// TIA Portal V20 export
// export: Created 2025-12-01T14:57:27.4021736Z, ExportSetting None, DisplayName Totally Integrated Automation Portal, DisplayVersion V20 Update 3, DisplayName TIA Portal Openness, DisplayVersion V20 Update 3, DisplayName TIA Portal Version Control Interface, DisplayVersion V20 Update 3, DisplayName STEP 7 Professional, DisplayVersion V20 Update 3, DisplayName STEP 7 Safety, DisplayVersion V20 Update 2, DisplayName WinCC Basic/Comfort/Advanced, DisplayVersion V20 Update 3, DisplayName WinCC Professional, DisplayVersion V20 Update 3, DisplayName WinCC Unified, DisplayVersion V20 Update 3
FUNCTION_BLOCK "FB607_SalidaMovil_Frontal_Quimarox"   // FB607, LAD
{ S7_Optimized_Access := 'FALSE' }
// stored: AutoNumber false, SetENOAutomatically false
   VAR_INPUT
      MesaDeDescarga : UInt;
      ID_Quimarox : UInt;
      ID_Elemento : UInt;
      DestinoAsociado : UInt;
      pHs_PosicionDescarga : Bool;
      pHs_Protrusion : Bool;
      En_PosicionReposo : Bool;
      Corte_PosicionReposo : Bool;
      Corte_PosicionDesCarga : Bool;
      En_PosicionDescarga : Bool;
      Permiso_DeDesCarga : Bool;
      V_Filtro_pHsPresencia : Int;
      Pto_Ajuste_1 : Int;   // en mm (paso a lenta en posicionamiento a descarga de transportador)
      Pto_Ajuste_2 : Int;   // en mm (timeout movimiento posicion descarga del transportador)
      Pto_Ajuste_3 : Int;   // en mm (paso a lenta en posicionamiento reposo del transportador)
      Pto_Ajuste_4 : Int;   // en mm (timeout movimiento posicion reposo del transportador)
   END_VAR
   VAR_OUTPUT
      NXT_DescargaActiva : Bool;
      ElevadorEnLenta : Bool;
      PararElevador : Bool;
      Ir_PosicionReposo : Bool;
      Ir_PosicionDescarga : Bool;
   END_VAR
   VAR
      FILTRO_pHsPresencia : "FB910_CNT_UHS";
      EstadoAsociadoEnMesa : UInt;
      Ultimo_PeineTratado : UInt;
      Aux_PeineEnDesCarga { ExternalAccessible := 'False'; ExternalVisible := 'False'; ExternalWritable := 'False'} : UInt;
   END_VAR
   VAR_TEMP
      MesaQuimarox : UInt;
      NumeroUT : UInt;
      Vagon_Siguiente : Int;
      EsMesaTL : Bool;
      FILTRO_PosicionDesCarga : Bool;
   END_VAR
BEGIN

NETWORK
TITLE = ERROR - Rearme
/////////////////////////////////////////////////////////////
/////////////////////////////////////////////////////////////
/////////////////////////////////////////////////////////////
// Rearne de Errores
      SET;
      A     "DB902_Estado_ZonaMesa".EstadoMesas[#MesaDeDescarga].Rearme_CBx;
      O     "DB902_Estado_ZonaMesa".EstadoMesas[#MesaDeDescarga].PerReset_CBx;
      R     "DB900_Estado_Mesas".EstadoVI[#MesaDeDescarga].Error_Mx;
      R     "DB900_Estado_Mesas".EstadoVI[#MesaDeDescarga].Err_Protusion;
      R     "DB900_Estado_Mesas".EstadoVI[#MesaDeDescarga].Err_TOut_Avance_E1_E3;
      R     "DB900_Estado_Mesas".EstadoVI[#MesaDeDescarga].Err_Tout_Sacar;
      R     "DB900_Estado_Mesas".EstadoVI[#MesaDeDescarga].Err_Tout_Recoger;

      R     "DB900_Estado_Mesas".EstadoVI[#MesaDeDescarga].Err_DatosPLC;



NETWORK
TITLE = HMI - Entradas y Salidas de la Mesa
/////////////////////////////////////////////////////////////
/////////////////////////////////////////////////////////////
/////////////////////////////////////////////////////////////
// Entradas
      SET;
      A     #pHs_PosicionDescarga;
      =     "DB904_Estado_Maquinas".EstadoVI[#MesaDeDescarga].Byte7_bit4;
      SET;
      A     #pHs_Protrusion;
      =     "DB904_Estado_Maquinas".EstadoVI[#MesaDeDescarga].Byte9_bit0;

      SET;
      A     #En_PosicionReposo;
      =     "DB904_Estado_Maquinas".EstadoVI[#MesaDeDescarga].Byte8_bit4;
      SET;
      A     #Corte_PosicionReposo;
      =     "DB904_Estado_Maquinas".EstadoVI[#MesaDeDescarga].Byte7_bit6;
      SET;
      A     #Corte_PosicionDesCarga;
      =     "DB904_Estado_Maquinas".EstadoVI[#MesaDeDescarga].Byte7_bit7;
      SET;
      A     #En_PosicionDescarga;
      =     "DB904_Estado_Maquinas".EstadoVI[#MesaDeDescarga].Byte8_bit5;


// Salidas
      SET;
      A     #NXT_DescargaActiva;
      =     "DB900_Estado_Mesas".EstadoVI[#MesaDeDescarga].Sa_Giro_180;
      SET;
      A     #Ir_PosicionReposo;
      =     "DB900_Estado_Mesas".EstadoVI[#MesaDeDescarga].Sa_Trans_Baj;
      SET;
      A     #Ir_PosicionDescarga;
      =     "DB900_Estado_Mesas".EstadoVI[#MesaDeDescarga].Sa_Trans_Sub;



NETWORK
TITLE = Comprobacion de que la MESA es de TRACKING
/////////////////////////////////////////////////////////////////////////////////////
/////////////////////////////////////////////////////////////////////////////////////
/////////////////////////////////////////////////////////////////////////////////////
// Comprobar si es una Mesa de Tracking o Routing
      SET;
      A     "DB850_DefinicionMesas".Mesa[#MesaDeDescarga].ConfigMesa.MesaTL;
      =     #EsMesaTL;



NETWORK
TITLE = Inicializacio PREVIA
/////////////////////////////////////////////////////////////////////////////////////
/////////////////////////////////////////////////////////////////////////////////////
/////////////////////////////////////////////////////////////////////////////////////
      CLR;
      =     #ElevadorEnLenta;
      =     #PararElevador;

      CLR;
      =     #NXT_DescargaActiva;

      CLR;
      =     #Ir_PosicionReposo;
      =     #Ir_PosicionDescarga;



NETWORK
TITLE = SISTEMA - Reset
/////////////////////////////////////////////////////////////
/////////////////////////////////////////////////////////////
/////////////////////////////////////////////////////////////
// - Existe RESET ??
      SET;
      AN    "DB902_Estado_ZonaMesa".EstadoMesas[#MesaDeDescarga].PerReset_CBx;  //#Estado_CBx.PerReset_CBx
      JC    NoRealizandose_Reset;

      L     0;
      T     #EstadoAsociadoEnMesa;
      T     #Ultimo_PeineTratado;


/////////////////////////////////////////////////////////////
/////////////////////////////////////////////////////////////
/////////////////////////////////////////////////////////////
// - Final Tratamiento del RESET
NoRealizandose_Reset:NOP   0;



NETWORK
TITLE = >>>>>>>>>>>>>>>>>>>>>>>>>>>>>>>>>>>>>>>>>>>>>>>>>>>>>>>>>>>>>>>>>>>

REGION Network 7: FILTRO - pHs de Presencia
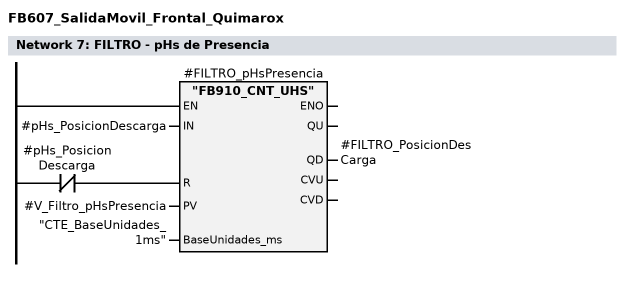
   RUNG wire#powerrail
      #FILTRO_pHsPresencia(R := wire#w1, IN := #pHs_PosicionDescarga, PV := #V_Filtro_pHsPresencia, BaseUnidades_ms := "CTE_BaseUnidades_1ms", QU =>, QD => #FILTRO_PosicionDesCarga, CVU =>, CVD =>)
   END_RUNG
   RUNG wire#powerrail
      I_Contact( #pHs_PosicionDescarga )
   END_RUNG wire#w1
   // the same network as SCL:
   #FILTRO_pHsPresencia(IN := #pHs_PosicionDescarga,   // "FB910_CNT_UHS"
                        R := NOT #pHs_PosicionDescarga,
                        PV := #V_Filtro_pHsPresencia,
                        BaseUnidades_ms := "CTE_BaseUnidades_1ms",
                        QD => #FILTRO_PosicionDesCarga);
END_REGION

NETWORK
TITLE = >>>>>>>>>>>>>>>>>>>>>>>>>>>>>>>>>>>>>>>>>>>>>>>>>>>>>>>>>>>>>>>>>>>

NETWORK
TITLE = Control Etapa activa >>> DISTRIBUCION
/////////////////////////////////////////////////////////////////////////////////////
/////////////////////////////////////////////////////////////////////////////////////
/////////////////////////////////////////////////////////////////////////////////////
// listado de saltos de programa
      L     #EstadoAsociadoEnMesa;

      JL    ETAPA_PorDefecto;
      JU    ETAPA_00_EnReset;
      JU    ETAPA_01_EnReposo;

      JU    ETAPA_02_EsperaPermisoDeDescarga;
      JU    ETAPA_03_MoverPosicionDescarga;
      JU    ETAPA_04_PreparadoParaDescarga;
      JU    ETAPA_05_FinDescarga;
      JU    ETAPA_06_MoverPosicionReposo;

      JU    ETAPA_PorDefecto;
      JU    ETAPA_PorDefecto;
      JU    ETAPA_PorDefecto;

      JU    ETAPA_10_ResetVacio_EsperaDesCargaDePeine;
      JU    ETAPA_11_ResetVacio_RecogerCargaDePeine;
      JU    ETAPA_12_ResetVacio_MoverPosicionReposo;
      JU    ETAPA_13_ResetCargado_EsperaPermisoDeDesCarga;
      JU    ETAPA_14_ResetCargado_MoverPosicionReposo;

ETAPA_PorDefecto:JU    FinFuncion;




NETWORK
TITLE = ETAPA 00 >>> En Reset
/////////////////////////////////////////////////////////////////////////////////////
/////////////////////////////////////////////////////////////////////////////////////
/////////////////////////////////////////////////////////////////////////////////////
ETAPA_00_EnReset:NOP   0;
      CLR;
      =     #Ir_PosicionReposo;
      =     #Ir_PosicionDescarga;

/////////////////////////////////////////////////////////////////////////////////////
// error de protusion
      SET;
      AN    #pHs_Protrusion;
      JC    ErrorProtrusion;

/////////////////////////////////////////////////////////////////////////////////////
// Tiene que estar en Marcha y Sin Error para continuar
      SET;
      AN    "DB902_Estado_ZonaMesa".EstadoMesas[#MesaDeDescarga].Marcha_CBx;
      O     "DB902_Estado_ZonaMesa".EstadoMesas[#MesaDeDescarga].Error_CBx;
      JC    ET00_PararElevador;


/////////////////////////////////////////////////////////////////////////////////////
// En Resposo
      SET;
      A     #En_PosicionReposo;
      JC    ET00_IrEtapa_01_EnReposo;


/////////////////////////////////////////////////////////////////////////////////////
// NO Reposo - Vacio
      SET;
      AN    #FILTRO_PosicionDesCarga;
      JC    ET00_Reset_10_ResetVacio_EsperaDesCargaDePeine;

/////////////////////////////////////////////////////////////////////////////////////
// NO Reposo - Con Carga
      SET;
      A     #FILTRO_PosicionDesCarga;
      JC    ET00_Reset_13_ResetCargado_EsperaPermisoDeDesCarga;


/////////////////////////////////////////////////////////////////////////////////////
// Final del Reparto  ?????? No DEBE LLEGAR AQUI
      BE;




/////////////////////////////////////////////////////////////////////////////////////
/////////////////////////////////////////////////////////////////////////////////////
/////////////////////////////////////////////////////////////////////////////////////
ET00_PararElevador:NOP   0;
      SET;
      =     #PararElevador;
      BE;


/////////////////////////////////////////////////////////////////////////////////////
/////////////////////////////////////////////////////////////////////////////////////
/////////////////////////////////////////////////////////////////////////////////////
ET00_IrEtapa_01_EnReposo:NOP   0;
      L     1;
      T     #EstadoAsociadoEnMesa;
      JU    ETAPA_01_EnReposo;


/////////////////////////////////////////////////////////////////////////////////////
/////////////////////////////////////////////////////////////////////////////////////
/////////////////////////////////////////////////////////////////////////////////////
ET00_Reset_10_ResetVacio_EsperaDesCargaDePeine:NOP   0;
      L     10;
      T     #EstadoAsociadoEnMesa;
      JU    ETAPA_10_ResetVacio_EsperaDesCargaDePeine;


/////////////////////////////////////////////////////////////////////////////////////
/////////////////////////////////////////////////////////////////////////////////////
/////////////////////////////////////////////////////////////////////////////////////
ET00_Reset_13_ResetCargado_EsperaPermisoDeDesCarga:NOP   0;
      L     13;
      T     #EstadoAsociadoEnMesa;
      JU    ETAPA_13_ResetCargado_EsperaPermisoDeDesCarga;



NETWORK
TITLE = ETAPA 01 >>> En Reposo
/////////////////////////////////////////////////////////////////////////////////////
/////////////////////////////////////////////////////////////////////////////////////
/////////////////////////////////////////////////////////////////////////////////////
// Estado de reposo esperando a que llegue una carga para este destino
ETAPA_01_EnReposo:NOP   0;
      SET;
      AN    #En_PosicionReposo;
      JC    ET01_IrEtapa_14_MoverPosicionReposo;

/////////////////////////////////////////////////////////////////////////////////////
// miramos si ya hemos comprobado el peine que está delante nuestro
      SET;
      L     "DB602_ElementosQuimarox".Quimarox[#ID_Quimarox].Elementos[#ID_Elemento].Numero_carrier;
      L     #Ultimo_PeineTratado;
      ==I;
      JC    ET01_SinPeineEnVentana;

/////////////////////////////////////////////////////////////////////////////////////
// si no hemos comprobado el peine, comprobamos si tenemos un peine en ventana
      SET;
      AN    "DB602_ElementosQuimarox".Quimarox[#ID_Quimarox].Elementos[#ID_Elemento].Hay_Carrier_en_ventana;
      JC    ET01_SinPeineEnVentana;

/////////////////////////////////////////////////////////////////////////////////////
// si no ha saltado es porque el carrier está en ventana. Comprobamos si es para nosotros
      L     "DB602_ElementosQuimarox".Quimarox[#ID_Quimarox].Elementos[#ID_Elemento].Numero_carrier;
      T     #Aux_PeineEnDesCarga;

      SET;
      L     "DB601_PeinesQuimarox".Quimarox[#ID_Quimarox].vagon[#Aux_PeineEnDesCarga].Destino_principal;
      L     #DestinoAsociado;
      ==I;
      JC    ET01_PeineParaLaMesa;

/////////////////////////////////////////////////////////////////////////////////////
// si no es para mi, me guardo que he chequeado el peine para no volver a comprobarlo
      L     "DB602_ElementosQuimarox".Quimarox[#ID_Quimarox].Elementos[#ID_Elemento].Numero_carrier;
      T     #Ultimo_PeineTratado;
      BE;


/////////////////////////////////////////////////////////////////////////////////////
/////////////////////////////////////////////////////////////////////////////////////
/////////////////////////////////////////////////////////////////////////////////////
ET01_SinPeineEnVentana:NOP   0;
      SET;  // Esta TOTALMENTE libre ?
      A(;
      O     #FILTRO_PosicionDesCarga;
      ON    #pHs_Protrusion;
      );
      JCN   FinFuncion;
      JU    ErrorProtrusion;


/////////////////////////////////////////////////////////////////////////////////////
/////////////////////////////////////////////////////////////////////////////////////
/////////////////////////////////////////////////////////////////////////////////////
ET01_PeineParaLaMesa:NOP   0;
      L     2;
      T     #EstadoAsociadoEnMesa;
      L     "DB602_ElementosQuimarox".Quimarox[#ID_Quimarox].Elementos[#ID_Elemento].Numero_carrier;
      T     #Ultimo_PeineTratado;

      JU    ETAPA_02_EsperaPermisoDeDescarga;


/////////////////////////////////////////////////////////////////////////////////////
/////////////////////////////////////////////////////////////////////////////////////
/////////////////////////////////////////////////////////////////////////////////////
ET01_IrEtapa_14_MoverPosicionReposo:NOP   0;
      L     14;
      T     #EstadoAsociadoEnMesa;
      JU    ETAPA_14_ResetCargado_MoverPosicionReposo;


NETWORK
TITLE = ETAPA 02 >>> Etapa Espera de Permiso de Descarga
/////////////////////////////////////////////////////////////////////////////////////
/////////////////////////////////////////////////////////////////////////////////////
/////////////////////////////////////////////////////////////////////////////////////
// Espera a Permiso de Descarga. Antes de iniciar el Ciclo de Descarga
ETAPA_02_EsperaPermisoDeDescarga:NOP   0;
      SET;
      A     #Permiso_DeDesCarga;
      JC    ET02_IrEtapa_03_MoverPosicionDesCarga;

      SET;  // No se puede Iniciar el Ciclo
      =     #PararElevador;
      BE;

/////////////////////////////////////////////////////////////////////////////////////
// Esta el Permiso de Descarga >>> Activar Ciclo de Descarga
ET02_IrEtapa_03_MoverPosicionDesCarga:NOP   0;
      L     3;
      T     #EstadoAsociadoEnMesa;

      JU    ETAPA_03_MoverPosicionDescarga;



NETWORK
TITLE = ETAPA 03 >>> Mover a Posicion de Descarga
/////////////////////////////////////////////////////////////////////////////////////
/////////////////////////////////////////////////////////////////////////////////////
/////////////////////////////////////////////////////////////////////////////////////
// inicio del proceso de descarga
// antes de iniciar la descarga tenemos que colocar el transportador en la posicion de descarga
ETAPA_03_MoverPosicionDescarga:NOP   0;
      SET;
      A     #En_PosicionDescarga;
      JC    ET03_IrEtapa_04_PreparadoParaDesCarga;

/////////////////////////////////////////////////////////////////////////////////////
      SET;
      =     #Ir_PosicionDescarga;
      CLR;
      =     #Ir_PosicionReposo;

/////////////////////////////////////////////////////////////////////////////////////
// como estamos metiendo el transportador, tenemos que vigilar que no tarda demasiado en entrar
      L     "DB602_ElementosQuimarox".Quimarox[#ID_Quimarox].Elementos[#ID_Elemento].Avance_carrier;  // #datos_elemento.Avance_carrier
      L     #Pto_Ajuste_1;
      <=I;
      JC    ET03_VelocidadNormal;

      SET;
      =     #ElevadorEnLenta;

      L     "DB602_ElementosQuimarox".Quimarox[#ID_Quimarox].Elementos[#ID_Elemento].Avance_carrier;  //#datos_elemento.Avance_carrier
      L     #Pto_Ajuste_2;
      >=I;
      JC    ErrorMoverPosicionDescarga;  // error de movimiento al sacar el transportador

      BE;


/////////////////////////////////////////////////////////////////////////////////////
ET03_VelocidadNormal:CLR;
      =     #ElevadorEnLenta;
      BE;

/////////////////////////////////////////////////////////////////////////////////////
ET03_IrEtapa_04_PreparadoParaDesCarga:CLR;
      =     #Ir_PosicionDescarga;
      L     4;
      T     #EstadoAsociadoEnMesa;

      JU    ETAPA_04_PreparadoParaDescarga;



NETWORK
TITLE = ETAPA 04 >>> Etapa Preparado para el Proceso de Descarga
/////////////////////////////////////////////////////////////////////////////////////
/////////////////////////////////////////////////////////////////////////////////////
/////////////////////////////////////////////////////////////////////////////////////
// espera a la descarga activa
// antes de iniciar la descarga tenemos que esperar a ver el detector de la descarga
ETAPA_04_PreparadoParaDescarga:NOP   0;
      SET;
      =     #NXT_DescargaActiva;

      SET;
      A     #FILTRO_PosicionDesCarga;
      A     #pHs_Protrusion;
      JC    ET04_IrEtapa_05_FinDescarga;


/////////////////////////////////////////////////////////////////////////////////////
// tenemos que comprobar si seguimos en la ventana, sino nos retiramos
      SET;
      AN    #pHs_Protrusion;
      JC    ErrorProtrusion;

/////////////////////////////////////////////////////////////////////////////////////
      SET;
      A     "DB602_ElementosQuimarox".Quimarox[#ID_Quimarox].Elementos[#ID_Elemento].Hay_Carrier_en_ventana;
      JC    FinFuncion;


/////////////////////////////////////////////////////////////////////////////////////
      SET;
      AN    "DB602_ElementosQuimarox".Quimarox[#ID_Quimarox].Elementos[#ID_Elemento].Hay_Carrier_en_ventana;
      JC    ET04_IrEtapa_06_MoverPosicionReposo;

      BE;


/////////////////////////////////////////////////////////////////////////////////////
ET04_IrEtapa_06_MoverPosicionReposo:NOP   0;
      L     6;
      T     #EstadoAsociadoEnMesa;
      JU    ETAPA_06_MoverPosicionReposo;

/////////////////////////////////////////////////////////////////////////////////////
// si hemos visto el detector, es que nos tenemos que poner en el estado de descarga activa.
ET04_IrEtapa_05_FinDescarga:NOP   0;
      L     5;
      T     #EstadoAsociadoEnMesa;
      JU    ETAPA_05_FinDescarga;



NETWORK
TITLE = ETAPA 05 >>> Fin Descarga
/////////////////////////////////////////////////////////////////////////////////////
/////////////////////////////////////////////////////////////////////////////////////
/////////////////////////////////////////////////////////////////////////////////////
// antes de saltar al inicio proceso reposo, vamos a ver si el siguiente peine que va a llegar
// tiene también una carga para nosotros. Para eso tenemos que sacar el dato del peine siguiente.
ETAPA_05_FinDescarga:NOP   0;
      SET;
      =     #NXT_DescargaActiva;

/////////////////////////////////////////////////////////////////////////////////////
/////////////////////////////////////////////////////////////////////////////////////
/////////////////////////////////////////////////////////////////////////////////////
// COMPROBAR EL TIPO DE MESA
      L     "CTE_Evento_QDES";
      T     "DB601_PeinesQuimarox".Quimarox[#ID_Quimarox].vagon[#Aux_PeineEnDesCarga].EventoAGenerar;
      L     #MesaDeDescarga;
      L     "CTE_OffsetMesa";
      +I;
      T     "DB601_PeinesQuimarox".Quimarox[#ID_Quimarox].vagon[#Aux_PeineEnDesCarga].Mesa_descarga;

      SET;
      AN    #EsMesaTL;
      JC    TRACKING_PasoDeDatos;
      JU    ROUTING_PasoDeDatos;

/////////////////////////////////////////////////////////////////////////////////////
// MESA DE ROUTING
ROUTING_PasoDeDatos:NOP   0;
      JU    FINAL_PasoDeDatos;

/////////////////////////////////////////////////////////////////////////////////////
// MESA DE TRACKING
// ANTES DE CREAR LA UT, TENGO QUE COMPROBAR SI EL MCKEY ES 0
TRACKING_PasoDeDatos:NOP   0;
      SET;
      L     "DB601_PeinesQuimarox".Quimarox[#ID_Quimarox].vagon[#Aux_PeineEnDesCarga].DatosCarga.Mckey;
      L     0;
      ==D;
      JC    TRACKING_CrearNueva_UT;

/////////////////////////////////////////////////////////////////////////////////////
// AQUI GENERAMOS LA UT EN LA MESA DE DESTINO CON MCKEY CONOCIDO
      CALL  "FC721_CrearUT_EnMesa"
      ( McKey      := "DB601_PeinesQuimarox".Quimarox[#ID_Quimarox].vagon[#Aux_PeineEnDesCarga].DatosCarga.Mckey,
        MesaActual := #MesaDeDescarga,
        NumeroUT   := #NumeroUT
      );

      L     11;  // Cambio de Mesa de la UT
      T     "DB812_UTs_Control".UT[#NumeroUT].EstadoEmisionUT;

      L     "DB601_PeinesQuimarox".Quimarox[#ID_Quimarox].vagon[#Aux_PeineEnDesCarga].DatosCarga.MesaDestino;
      T     "DB812_UTs_Control".UT[#NumeroUT].MesaDestino;
      T     "DB813_UTs_Ruta".UT[#NumeroUT].Ruta[0];

      JU    FINAL_PasoDeDatos;

/////////////////////////////////////////////////////////////////////////////////////
// AQUI GENERAMOS LA UT EN LA MESA DE DESTINO CON MCKEY DESCONOCIDO
TRACKING_CrearNueva_UT:NOP   0;
      CALL  "FC723_InsertarUT_EnMesa"
      ( MesaActual := #MesaDeDescarga,
        NumeroUT   := #NumeroUT
      );

      L     12;  // Aviso de Nueva UT en la Mesa
      T     "DB812_UTs_Control".UT[#NumeroUT].EstadoEmisionUT;

      JU    FINAL_PasoDeDatos;


/////////////////////////////////////////////////////////////////////////////////////
/////////////////////////////////////////////////////////////////////////////////////
/////////////////////////////////////////////////////////////////////////////////////
FINAL_PasoDeDatos:NOP   0;
      L     6;
      T     #EstadoAsociadoEnMesa;
      JU    ETAPA_06_MoverPosicionReposo;



NETWORK
TITLE = ETAPA 06 >>> Mover a Posicion de Reposo
/////////////////////////////////////////////////////////////////////////////////////
/////////////////////////////////////////////////////////////////////////////////////
/////////////////////////////////////////////////////////////////////////////////////
// inicio del proceso de vuelta a reposo
ETAPA_06_MoverPosicionReposo:NOP   0;
      CLR;
      =     #NXT_DescargaActiva;

      SET;
      A     #En_PosicionReposo;
      JC    ET06_REPOSO_IrEtapa_01_EnReposo;

/////////////////////////////////////////////////////////////////////////////////////
      SET;
      =     #Ir_PosicionReposo;

      L     "DB602_ElementosQuimarox".Quimarox[#ID_Quimarox].Elementos[#ID_Elemento].Avance_carrier;  //#datos_elemento.Avance_carrier
      L     #Pto_Ajuste_3;
      <=I;
      JC    ET06_REPOSO_VelocidadNormal;

      SET;
      =     #ElevadorEnLenta;

/////////////////////////////////////////////////////////////////////////////////////
      SET;
      L     "DB602_ElementosQuimarox".Quimarox[#ID_Quimarox].Elementos[#ID_Elemento].Avance_carrier;  // #datos_elemento.Avance_carrier
      L     #Pto_Ajuste_4;
      >=I;
      JC    ErrorMoverPosicionReposo;  // error de movimiento al meter el transportador

/////////////////////////////////////////////////////////////////////////////////////
      SET;
      AN    "DB602_ElementosQuimarox".Quimarox[#ID_Quimarox].Elementos[#ID_Elemento].Hay_Carrier_en_ventana;  //#datos_elemento.Hay_Carrier_en_ventana
      JC    ErrorMoverPosicionReposo;

      BE;

/////////////////////////////////////////////////////////////////////////////////////
ET06_REPOSO_VelocidadNormal:NOP   0;
      CLR;
      =     #ElevadorEnLenta;
      BE;

/////////////////////////////////////////////////////////////////////////////////////
ET06_REPOSO_IrEtapa_01_EnReposo:NOP   0;
      CLR;
      =     #Ir_PosicionReposo;
      =     #ElevadorEnLenta;

      L     1;
      T     #EstadoAsociadoEnMesa;
      BE;



NETWORK
TITLE = >>>>>>>>>>>>>>>>>>>>>>>>>>>>>>>>>>>>>>>>>>>>>>>>>>>>>>>>>>>>>>>>>>>

NETWORK
TITLE = ETAPA 10 >>> RESET VACIO - EsperaDesCarga del Peine
/////////////////////////////////////////////////////////////////////////////////////
/////////////////////////////////////////////////////////////////////////////////////
/////////////////////////////////////////////////////////////////////////////////////
// Mirar si el peine Actal Existe Carga para el elemento
ETAPA_10_ResetVacio_EsperaDesCargaDePeine:NOP   0;
      SET;
      =     #PararElevador;


/////////////////////////////////////////////////////////////////////////////////////
// error de protusion
      SET;
      AN    #pHs_Protrusion;
      JC    ErrorProtrusion;

/////////////////////////////////////////////////////////////////////////////////////
// si no hemos comprobado el peine, comprobamos si tenemos un peine en ventana
      SET;
      AN    "DB602_ElementosQuimarox".Quimarox[#ID_Quimarox].Elementos[#ID_Elemento].Hay_Carrier_en_ventana;
      JC    ET10_RESET_IrEtapa_12_MoverPosicionReposo;

/////////////////////////////////////////////////////////////////////////////////////
// Comprobamos si es para nosotros, El peine
      L     "DB602_ElementosQuimarox".Quimarox[#ID_Quimarox].Elementos[#ID_Elemento].Numero_carrier;
      T     #Aux_PeineEnDesCarga;

      SET;
      L     "DB601_PeinesQuimarox".Quimarox[#ID_Quimarox].vagon[#Aux_PeineEnDesCarga].Destino_principal;
      L     #DestinoAsociado;
      ==I;
      JC    ET10_RESET_IrEtapa_11_RecogerCargaDePeine;

/////////////////////////////////////////////////////////////////////////////////////
// si no es para mi, me guardo que he chequeado el peine para no volver a comprobarlo
      L     "DB602_ElementosQuimarox".Quimarox[#ID_Quimarox].Elementos[#ID_Elemento].Numero_carrier;
      T     #Ultimo_PeineTratado;

      JU    ET10_RESET_IrEtapa_12_MoverPosicionReposo;


/////////////////////////////////////////////////////////////////////////////////////
/////////////////////////////////////////////////////////////////////////////////////
/////////////////////////////////////////////////////////////////////////////////////
ET10_RESET_IrEtapa_11_RecogerCargaDePeine:NOP   0;

      L     "DB602_ElementosQuimarox".Quimarox[#ID_Quimarox].Elementos[#ID_Elemento].Numero_carrier;
      T     #Ultimo_PeineTratado;

      L     11;
      T     #EstadoAsociadoEnMesa;
      JU    ETAPA_11_ResetVacio_RecogerCargaDePeine;

/////////////////////////////////////////////////////////////////////////////////////
/////////////////////////////////////////////////////////////////////////////////////
/////////////////////////////////////////////////////////////////////////////////////
ET10_RESET_IrEtapa_12_MoverPosicionReposo:NOP   0;
      L     "DB602_ElementosQuimarox".Quimarox[#ID_Quimarox].Elementos[#ID_Elemento].Numero_carrier;
      T     #Ultimo_PeineTratado;

      L     12;
      T     #EstadoAsociadoEnMesa;
      JU    ETAPA_12_ResetVacio_MoverPosicionReposo;



NETWORK
TITLE = ETAPA 11 >>> RESET VACIO - Recoger Carga Del Peine
/////////////////////////////////////////////////////////////////////////////////////
/////////////////////////////////////////////////////////////////////////////////////
/////////////////////////////////////////////////////////////////////////////////////
// Recoger la Carga a Velocidad Lenta por SEGURIDAD
// Deberia descargar SIEMPE >>> SINO NO PASAR AQUI
ETAPA_11_ResetVacio_RecogerCargaDePeine:NOP   0;
      SET;
      =     #ElevadorEnLenta;

/////////////////////////////////////////////////////////////////////////////////////
      SET;
      AN    #Permiso_DeDesCarga;
      JC    ET11_PararElevador;


/////////////////////////////////////////////////////////////////////////////////////
      SET;
      =     #NXT_DescargaActiva;

      SET;
      A     #FILTRO_PosicionDesCarga;
      A     #pHs_Protrusion;
      JC    ET11_IrEtapa_5_FinDescarga;


/////////////////////////////////////////////////////////////////////////////////////
// Error de Carga
      SET;
      AN    #pHs_Protrusion;
      JC    ErrorProtrusion;

/////////////////////////////////////////////////////////////////////////////////////
// Si no esta en VENTADA --- ERROR
      SET;
      AN    "DB602_ElementosQuimarox".Quimarox[#ID_Quimarox].Elementos[#ID_Elemento].Hay_Carrier_en_ventana;
      JC    ErrorDatosCargada;

      BE;

/////////////////////////////////////////////////////////////////////////////////////
/////////////////////////////////////////////////////////////////////////////////////
/////////////////////////////////////////////////////////////////////////////////////
ET11_PararElevador:NOP   0;
      SET;
      =     #PararElevador;
      BE;


/////////////////////////////////////////////////////////////////////////////////////
/////////////////////////////////////////////////////////////////////////////////////
/////////////////////////////////////////////////////////////////////////////////////
// si hemos visto el detector, es que nos tenemos que poner en el estado de descarga activa.
ET11_IrEtapa_5_FinDescarga:NOP   0;
      L     5;
      T     #EstadoAsociadoEnMesa;
      JU    ETAPA_05_FinDescarga;




NETWORK
TITLE = ETAPA 12 >>> RESET VACIO - Mover Posicion Reposo
/////////////////////////////////////////////////////////////////////////////////////
/////////////////////////////////////////////////////////////////////////////////////
/////////////////////////////////////////////////////////////////////////////////////
// Mover a Posicion Reposo >>> NO ESPERA CARGA
ETAPA_12_ResetVacio_MoverPosicionReposo:NOP   0;
      SET;
      =     #Ir_PosicionReposo;
      =     #PararElevador;


/////////////////////////////////////////////////////////////////////////////////////
      SET;
      A     #En_PosicionReposo;
      JC    ET12_RESET_IrEtapa_01_EnReposo;

      BE;


/////////////////////////////////////////////////////////////////////////////////////
/////////////////////////////////////////////////////////////////////////////////////
/////////////////////////////////////////////////////////////////////////////////////
ET12_RESET_IrEtapa_01_EnReposo:NOP   0;
      CLR;
      =     #Ir_PosicionReposo;
      =     #PararElevador;

      L     1;
      T     #EstadoAsociadoEnMesa;
      JU    ETAPA_01_EnReposo;



NETWORK
TITLE = >>>>>>>>>>>>>>>>>>>>>>>>>>>>>>>>>>>>>>>>>>>>>>>>>>>>>>>>>>>>>>>>>>>

NETWORK
TITLE = ETAPA 13 >>> RESET CARGADO - Espera De Permiso De DesCarga
/////////////////////////////////////////////////////////////////////////////////////
/////////////////////////////////////////////////////////////////////////////////////
/////////////////////////////////////////////////////////////////////////////////////
// Espera a Permiso de Descarga.
ETAPA_13_ResetCargado_EsperaPermisoDeDesCarga:NOP   0;
      SET;
      =     #NXT_DescargaActiva;
      =     #PararElevador;

/////////////////////////////////////////////////////////////////////////////////////
      SET;
      A     #Permiso_DeDesCarga;
      JC    ET13_RESET_IrEtapa_14_MoverPosicionReposo;

      BE;


/////////////////////////////////////////////////////////////////////////////////////
/////////////////////////////////////////////////////////////////////////////////////
/////////////////////////////////////////////////////////////////////////////////////
// Esta el Permiso de Descarga
ET13_RESET_IrEtapa_14_MoverPosicionReposo:NOP   0;
      L     14;
      T     #EstadoAsociadoEnMesa;
      JU    ETAPA_14_ResetCargado_MoverPosicionReposo;



NETWORK
TITLE = ETAPA 14 >>> RESET CARGADO - Mover a Posicion de Reposo
/////////////////////////////////////////////////////////////////////////////////////
/////////////////////////////////////////////////////////////////////////////////////
/////////////////////////////////////////////////////////////////////////////////////
//
ETAPA_14_ResetCargado_MoverPosicionReposo:NOP   0;
      SET;
      =     #Ir_PosicionReposo;
      =     #PararElevador;

/////////////////////////////////////////////////////////////////////////////////////
      SET;
      A     #En_PosicionReposo;
      JC    ET14_RESET_IrEtapa_01_EnReposo;

      BE;


/////////////////////////////////////////////////////////////////////////////////////
/////////////////////////////////////////////////////////////////////////////////////
/////////////////////////////////////////////////////////////////////////////////////
ET14_RESET_IrEtapa_01_EnReposo:NOP   0;
      CLR;
      =     #Ir_PosicionReposo;
      =     #PararElevador;

      L     1;
      T     #EstadoAsociadoEnMesa;
      JU    ETAPA_01_EnReposo;



NETWORK
TITLE = >>>>>>>>>>>>>>>>>>>>>>>>>>>>>>>>>>>>>>>>>>>>>>>>>>>>>>>>>>>>>>>>>>>

NETWORK
TITLE = ERRRORES DE LA MESA >>> Activacion
/////////////////////////////////////////////////////////////////////////////////////
/////////////////////////////////////////////////////////////////////////////////////
/////////////////////////////////////////////////////////////////////////////////////
ErrorProtrusion:SET;
      =     #PararElevador;
      =     "DB900_Estado_Mesas".EstadoVI[#MesaDeDescarga].Error_Mx;
      =     "DB900_Estado_Mesas".EstadoVI[#MesaDeDescarga].Err_Protusion;
      BE;

/////////////////////////////////////////////////////////////////////////////////////
/////////////////////////////////////////////////////////////////////////////////////
/////////////////////////////////////////////////////////////////////////////////////
ErrorMoverPosicionDescarga:SET;
      =     #PararElevador;
      =     "DB900_Estado_Mesas".EstadoVI[#MesaDeDescarga].Error_Mx;
      =     "DB900_Estado_Mesas".EstadoVI[#MesaDeDescarga].Err_Tout_Sacar;
      BE;

/////////////////////////////////////////////////////////////////////////////////////
/////////////////////////////////////////////////////////////////////////////////////
/////////////////////////////////////////////////////////////////////////////////////
ErrorMoverPosicionReposo:SET;
      =     #PararElevador;
      =     "DB900_Estado_Mesas".EstadoVI[#MesaDeDescarga].Error_Mx;
      =     "DB900_Estado_Mesas".EstadoVI[#MesaDeDescarga].Err_Tout_Recoger;
      BE;

/////////////////////////////////////////////////////////////////////////////////////
/////////////////////////////////////////////////////////////////////////////////////
/////////////////////////////////////////////////////////////////////////////////////
ErrorDatosCargada:NOP   0;  // error en la carga
      SET;
      =     "DB900_Estado_Mesas".EstadoVI[#MesaDeDescarga].Error_Mx;
      =     "DB900_Estado_Mesas".EstadoVI[#MesaDeDescarga].Err_DatosPLC;
      =     #PararElevador;
      BE;



NETWORK
TITLE = FIN DE LA FUNCION
/////////////////////////////////////////////////////////////////////////////////////
/////////////////////////////////////////////////////////////////////////////////////
/////////////////////////////////////////////////////////////////////////////////////
FinFuncion:BE;


END_FUNCTION_BLOCK
